// LS Electric XG5000 project: xg
// PLC LSPLC
// module base 0 slot 0: 입출력 모듈:XBC-DR32H (DC 24V 입력, 릴레이 출력 32점)
// module base 0 slot 1: 위치결정 모듈:XBF-PD02A (위치결정 펄스(LD)출력형, 2축)
// module base 0 slot 2: 출력 모듈:XBE-TN/TP16A (트랜지스터 출력, 16점 (싱크출력/소스출력))

PROGRAM NewProgram (task: 스캔 프로그램)

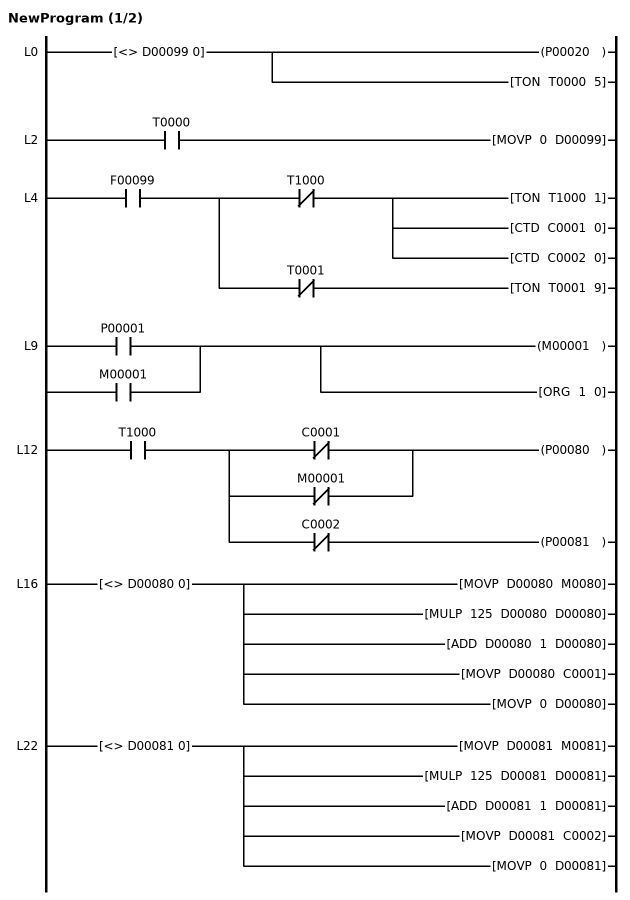
; L0
LOAD<>    D00099 0
OUT       P00020
TON       T0000 5
; L2
LOAD      T0000
MOVP      0 D00099
; L4
LOAD      F00099
MPUSH
AND NOT   T1000
TON       T1000 1
CTD       C0001 0
CTD       C0002 0
MPOP
AND NOT   T0001
TON       T0001 9
; L9
LOAD      P00001
OR        M00001
OUT       M00001
ORG       1 0
; L12
LOAD      T1000
MPUSH
LOAD NOT  C0001
OR NOT    M00001
AND LOAD
OUT       P00080
MPOP
AND NOT   C0002
OUT       P00081
; L16
LOAD<>    D00080 0
MOVP      D00080 M0080
MULP      125 D00080 D00080
ADD       D00080 1 D00080
MOVP      D00080 C0001
MOVP      0 D00080
; L22
LOAD<>    D00081 0
MOVP      D00081 M0081
MULP      125 D00081 D00081
ADD       D00081 1 D00081
MOVP      D00081 C0002
MOVP      0 D00081

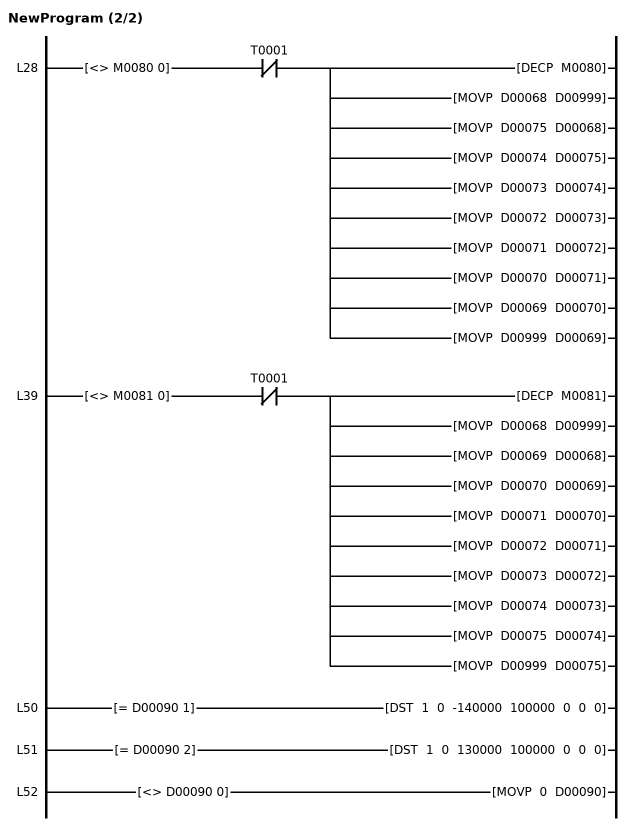
; L28
LOAD<>    M0080 0
AND NOT   T0001
DECP      M0080
MOVP      D00068 D00999
MOVP      D00075 D00068
MOVP      D00074 D00075
MOVP      D00073 D00074
MOVP      D00072 D00073
MOVP      D00071 D00072
MOVP      D00070 D00071
MOVP      D00069 D00070
MOVP      D00999 D00069
; L39
LOAD<>    M0081 0
AND NOT   T0001
DECP      M0081
MOVP      D00068 D00999
MOVP      D00069 D00068
MOVP      D00070 D00069
MOVP      D00071 D00070
MOVP      D00072 D00071
MOVP      D00073 D00072
MOVP      D00074 D00073
MOVP      D00075 D00074
MOVP      D00999 D00075
; L50
LOAD=     D00090 1
DST       1 0 -140000 100000 0 0 0
; L51
LOAD=     D00090 2
DST       1 0 130000 100000 0 0 0
; L52
LOAD<>    D00090 0
MOVP      0 D00090